Fanuc KAREL source: kt00641.KL

-- PROVISIONAL review KL for V770-1; original PC SHA256 e18d9ab5b644f7d2e4a9054e32ef3b0605955cee4c414922b2ad29bd122c260e
-- Incomplete behavior may be omitted. Consult companion uncertainty JSON. Do not deploy.
PROGRAM KT00641
%NOLOCKGROUP
VAR
  OUT : REAL
-- UNRESOLVED_DECL Y1 type=002018
-- UNRESOLVED_DECL Y2 type=002018
BEGIN
  -- UNRESOLVED_PC offsets 5-19; opcodes 2E,22,9D,33,B2
  -- UNRESOLVED_PC offsets 24-38; opcodes 2E,22,9D,33,B2
  -- UNRESOLVED_PC offsets 43-57; opcodes 2E,22,9D,33,B2
  -- UNRESOLVED_PC offsets 62-76; opcodes 2E,22,9D,33,B2
  -- UNRESOLVED_PC offsets 81-98; opcodes 22,9D,33,B1,51,64,23
  -- UNRESOLVED_PC offsets 103-107; opcodes 7F
END KT00641
